TYPE ST_TestStation_IN :
STRUCT
	bTestInput	: BOOL;
END_STRUCT
END_TYPE

(* stored: Version 1.1.0.1, ProductVersion 3.1.4020.12
   DUT ST_TestStation_IN: Id {fb48245f-6812-4227-8aaa-41fcda4cfeb0} *)
